{attribute 'qualified_only'}
{attribute 'strict'}
TYPE E_MachineMode :
(
	auto,
	manual, 
	none
);
END_TYPE

(* stored: Version 1.1.0.1, ProductVersion 3.1.4024.16
   DUT E_MachineMode: Id {889741ed-5150-423b-8cfe-e0adc246b8d8} *)
